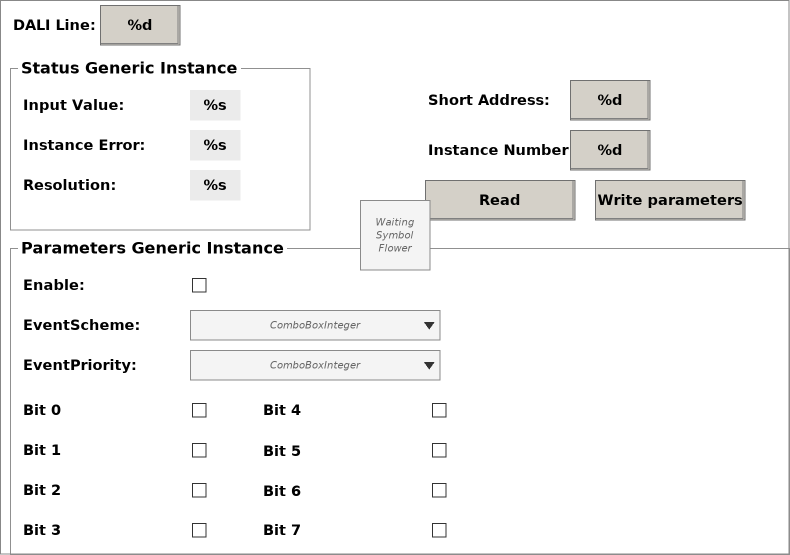
VISUALIZATION Visu_Part300GenericDevice  // 790x555
    GroupBox (10,240 780x315), "Parameters Generic Instance"
        Textfield (10,30 150x30), "Enable:"
        Checkbox (180,30 30x30), variable: DALI_Commissioning.fbPart300GenericDevice.bEnable
        Textfield (10,110 150x30), "EventPriority:"
        Textfield (10,195 100x30), "Bit 1"
        Textfield (10,155 100x30), "Bit 0"
        Checkbox (180,155 30x30), variable: DALI_Commissioning.fbPart300GenericDevice.bBit0
        Checkbox (180,195 30x30), variable: DALI_Commissioning.fbPart300GenericDevice.bBit1
        Textfield (10,235 100x30), "Bit 2"
        Textfield (250,155 100x30), "Bit 4"
        Textfield (250,196 100x30), "Bit 5"
        Checkbox (420,195 30x30), variable: DALI_Commissioning.fbPart300GenericDevice.bBit5
        Checkbox (420,155 30x30), variable: DALI_Commissioning.fbPart300GenericDevice.bBit4
        Checkbox (180,275 30x30), variable: DALI_Commissioning.fbPart300GenericDevice.bBit3
        Checkbox (180,235 30x30), variable: DALI_Commissioning.fbPart300GenericDevice.bBit2
        ComboBoxInteger (180,70 250x30), variable: DALI_Commissioning.fbPart300GenericDevice.eEventScheme, text list: 'EventScheme'
        Textfield (10,70 150x30), "EventScheme:"
        Textfield (250,236 100x30), "Bit 6"
        ComboBoxInteger (180,110 250x30), variable: DALI_Commissioning.fbPart300GenericDevice.eEventPriority, text list: 'EventPriority'
        Textfield (10,275 100x30), "Bit 3"
        Checkbox (420,235 30x30), variable: DALI_Commissioning.fbPart300GenericDevice.bBit6
        Checkbox (420,275 30x30), variable: DALI_Commissioning.fbPart300GenericDevice.bBit7
        Textfield (250,275 100x30), "Bit 7"
    GroupBox (10,60 300x170), "Status Generic Instance"
        Textfield (180,30 50x30), "%s", text variable: DALI_Commissioning.fbPart300GenericDevice.nInputValue
        Textfield (180,70 50x30), "%s", text variable: DALI_Commissioning.fbPart300GenericDevice.nInstanceError
        Textfield (180,110 50x30), "%s", text variable: DALI_Commissioning.fbPart300GenericDevice.nResolution
        Textfield (10,30 160x30), "Input Value:"
        Textfield (10,70 160x30), "Instance Error:"
        Textfield (10,110 160x30), "Resolution:"
    Button (425,180 150x40), "Read"
        OnMouseClick: execute { DALI_Commissioning.fbPart300GenericDevice.bRead := TRUE; }
    WaitingSymbolFlower (360,200 70x70), invisible if: DALI_Commissioning.fbPart300GenericDevice.bHideWaitSymbol
    Button (595,180 150x40), "Write parameters"
        OnMouseClick: execute { DALI_Commissioning.fbPart300GenericDevice.bWrite := TRUE; }
    Textfield (425,130 150x40), "Instance Number:"
    Textfield (425,80 150x40), "Short Address:"
    Button (570,80 80x40), "%d", text variable: DALI_Commissioning.fbPart300GenericDevice.nAddress
        OnMouseClick: write the text variable via Default, min 0, max 63, title "Insert Short Address"
    Button (570,130 80x40), "%d", text variable: DALI_Commissioning.fbPart300GenericDevice.nInstanceAddress
        OnMouseClick: write the text variable via Default, min 0, max 31, title "Insert instance number"
    Group (10,5 170x40)
        Textfield (0,0 110x40), "DALI Line:"
        Button (90,0 80x40), "%d", text variable: GVL_Internal.nDALILine
            OnMouseClick: write the text variable via Default, min 1, max 10, title "Choose line"
END_VISUALIZATION

(* stored: Version 1.1.0.1, ProductVersion 3.1.4024.12
   Visu Visu_Part300GenericDevice: Id {9f423c9c-f184-49dd-b64c-05d54423791b} *)
